FUNCTION_BLOCK FB_DancerControl
VAR_IN_OUT
	Master: AXIS_REF;
	Slave: AXIS_REF;
END_VAR
VAR_INPUT
	Enable: BOOL;
	/// Input signal for tension of the Web, usually represented by the relative actual dancer position senso 
	TensionInput: LREAL;
	/// Structure with Dancer Controller Parameter 
	Dancer_CTL: DANCER_REF;
END_VAR
VAR_OUTPUT
	Busy: BOOL;
	Error: BOOL;
	ErrorID: UDINT;
END_VAR
VAR
	state: E_DancerControlState := STATE_DANCERCONTROL_INITIALIZATION;
	GearInDyn: MC_GearInDyn;
	GearRatio: LREAL;
	InGear: BOOL;
	GearOut: MC_GearOut;
	ExecuteGearIn: BOOL;
	ExecuteGearOut: BOOL;
	PID: FB_BasicPID;
	CPUcounter: GETCPUCOUNTER;
	CPUcounter_LastLo: UDINT;
	CPUcounter_LastHi: UDINT;
	ControlCycleTime: LREAL;
	PIDoutput: LREAL;
	PIDerrorID: UDINT;
	Halt: MC_Halt;
	GetCurrentTaskIndex: GETCURTASKINDEX;
	AxisIsMoving: BOOL;
END_VAR

IF GetCurrentTaskIndex.index = 0 THEN
	(* get cycle time *)
	GetCurrentTaskIndex();
END_IF

ControlCycleTime := TwinCAT_SystemInfoVarList._TaskInfo[GetCurrentTaskIndex.index].cycleTime / 1E7;

CASE state OF
	STATE_DANCERCONTROL_INITIALIZATION:
		Busy := FALSE;
		ExecuteGearIn := FALSE;
		IF Enable THEN
			Busy := TRUE;
			ExecuteGearIn := TRUE;
			ExecuteGearOut := FALSE;
			ActDancerControlPID();  (* FB_BasicPID *)
			PID(bReset:=TRUE);
			GearRatio := Dancer_CTL.deltaGear * PID.fCtrlOutput + Dancer_CTL.GearOffset;
			Dancer_CTL.GearRatio := GearRatio;
			Error := PIDerrorID<>0;
			IF Error THEN
				ErrorID := SEL(PIDerrorID=1, PIDerrorID, DANCERCONTROL_ERROR_INVALID_PID_PARAMETER );
				ErrorID := SEL(PIDerrorID=2, PIDerrorID, DANCERCONTROL_ERROR_INVALID_CYCLETIME );
				state := STATE_DANCERCONTROL_ERROR;
			ELSE
				state := STATE_DANCERCONTROL_ORDER;
			END_IF
		END_IF

	STATE_DANCERCONTROL_ORDER:
		IF GearInDyn.CommandAborted OR GearInDyn.Error OR NOT Enable THEN
			Error := GearInDyn.Error;
			ErrorID := GearInDyn.ErrorID;
			ExecuteGearIn := FALSE;
			ExecuteGearOut := TRUE;
			state := STATE_DANCERCONTROL_STOP;
		ELSIF Enable AND InGear THEN
			state := STATE_DANCERCONTROL_RUNNING;
		END_IF

	STATE_DANCERCONTROL_WAITING:
		IF GearInDyn.CommandAborted OR GearInDyn.Error OR NOT Enable THEN
			Error := GearInDyn.Error;
			ErrorID := GearInDyn.ErrorID;
			ExecuteGearIn := FALSE;
			ExecuteGearOut := TRUE;
			state := STATE_DANCERCONTROL_STOP;
		ELSIF Enable AND Master.Status.Moving THEN
			state := STATE_DANCERCONTROL_RUNNING;
		END_IF

	STATE_DANCERCONTROL_RUNNING:
		IF GearInDyn.CommandAborted OR GearInDyn.Error OR NOT Enable THEN
			Error := GearInDyn.Error;
			ErrorID := GearInDyn.ErrorID;
			ExecuteGearIn := FALSE;
			ExecuteGearOut := TRUE;
			state := STATE_DANCERCONTROL_STOP;
		ELSIF Enable AND Master.Status.Moving THEN
			(* active state *)
			ActDancerControlPID();
			GearRatio := Dancer_CTL.deltaGear * PID.fCtrlOutput + Dancer_CTL.GearOffset;
			Dancer_CTL.GearRatio := GearRatio;
		ELSE
			state := STATE_DANCERCONTROL_WAITING;
		END_IF

	STATE_DANCERCONTROL_STOP:
		ExecuteGearOut := TRUE;
		IF Halt.Done THEN
			GearRatio := 0;
			Dancer_CTL.GearRatio := 0;
			state := STATE_DANCERCONTROL_INITIALIZATION;
		ELSIF GearOut.Error THEN
			Error := GearOut.Error;
			ErrorID := GearOut.ErrorID;
			GearRatio := 0;
			Dancer_CTL.GearRatio := 0;
			state := STATE_DANCERCONTROL_ERROR;
		ELSIF Halt.Error THEN
			Error := Halt.Error;
			ErrorID := Halt.ErrorID;
			GearRatio := 0;
			Dancer_CTL.GearRatio := 0;
			state := STATE_DANCERCONTROL_ERROR;
		END_IF

	STATE_DANCERCONTROL_ERROR:
		Error := TRUE;
		Busy := FALSE;
		IF NOT Enable THEN
			state := STATE_DANCERCONTROL_INITIALIZATION;
		END_IF

ELSE
	(* unknown program state *)
	state := STATE_DANCERCONTROL_INITIALIZATION;
END_CASE

(* call actions *)
ActDancerControlGearIn();

IF state = STATE_DANCERCONTROL_INITIALIZATION THEN
	Busy := FALSE; (* reset busy as soon as possible *)
END_IF

ACTION ActDancerControlGearIn:
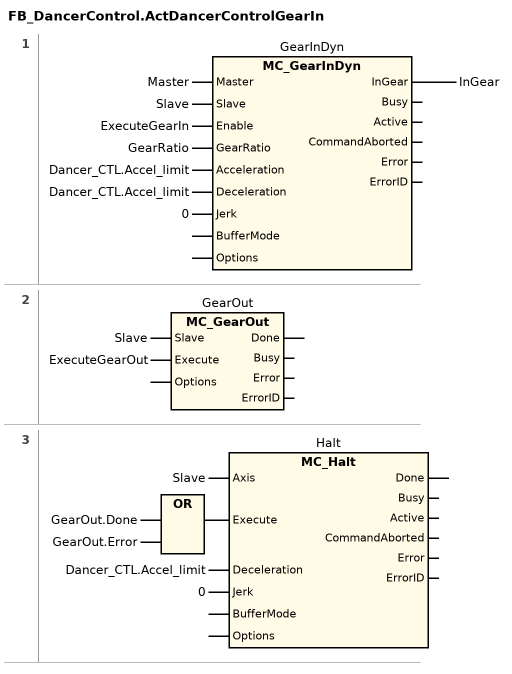
// NETWORK 1
GearInDyn(
    Master := Master,
    Slave := Slave,
    Enable := ExecuteGearIn,
    GearRatio := GearRatio,
    Acceleration := Dancer_CTL.Accel_limit,
    Deceleration := Dancer_CTL.Accel_limit,
    Jerk := 0); // MC_GearInDyn
InGear := GearInDyn.InGear;

// NETWORK 2
GearOut(Slave := Slave, Execute := ExecuteGearOut); // MC_GearOut

// NETWORK 3
Halt(
    Axis := Slave,
    Execute := GearOut.Done OR GearOut.Error,
    Deceleration := Dancer_CTL.Accel_limit,
    Jerk := 0); // MC_Halt
END_ACTION

ACTION ActDancerControlPID:
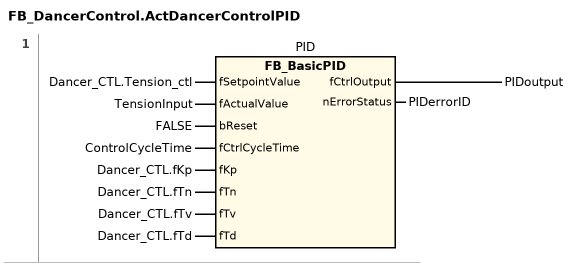
// NETWORK 1
PID(
    fSetpointValue := Dancer_CTL.Tension_ctl,
    fActualValue := TensionInput,
    bReset := FALSE,
    fCtrlCycleTime := ControlCycleTime,
    fKp := Dancer_CTL.fKp,
    fTn := Dancer_CTL.fTn,
    fTv := Dancer_CTL.fTv,
    fTd := Dancer_CTL.fTd,
    nErrorStatus => PIDerrorID); // FB_BasicPID
PIDoutput := PID.fCtrlOutput;
END_ACTION

END_FUNCTION_BLOCK

(* stored: Version 1.1.0.1, ProductVersion 3.1.4024.11
   POU FB_DancerControl: Id {9e2af623-efff-460f-a2a6-ddcefed0d78d}, SpecialFunc None
   Action ActDancerControlGearIn: Id {2270882d-ac02-4f6d-9876-a68345f7a2c2}
   Action ActDancerControlPID: Id {3d40e74a-132e-4014-8587-cb0287584e2f} *)
